# EPICS autosave request: devel/iocBoot/sioc-esb-avac01/aVac.req
$(P):CH1.DESC
$(P):CH2.DESC
$(P):CH3.DESC
$(P):CH4.DESC
